// TIA Portal project "Project_Timers_Sim" (V16)

(* hardware
DEVICE "S7-1200 station_1"  S7-1200 Station
   slot 0: "Rack_0"  S7-1200 Rack  Rack  V1.0
   slot 1: "PLC_1"  CPU 1212C DC/DC/Rly  6ES7 212-1HE40-0XB0  V4.4
*)

// ===== PLC "PLC_1"  CPU 1212C DC/DC/Rly =====

VAR_GLOBAL   // PLC tag table "Default tag table"
   ""START BUT"" AT %I0.0 : Bool;
   ""STOP BUT"" AT %I0.1 : Bool;
   ""MOTOR 1 KONT"" AT %Q0.0 : Bool;
   ""MOTOR 2 KONT"" AT %Q0.1 : Bool;
   ""MOTOR 3 KONT"" AT %Q0.2 : Bool;
END_VAR